(* This function Block interfaces with a NO turbo valve*)
(* Mainly used in the FEE HXR GATT*)
FUNCTION F_TurboExtILK_NO_1 : BOOL
VAR_INPUT
    Turbo		:	ST_PTM;
    BackingGauge:	ST_VG;
    InletGauge	:	ST_VG;
    VentValve	:	ST_VCC_NO; //NO type turbo valve
    ScrollPump	:	ST_RoughPump;
END_VAR

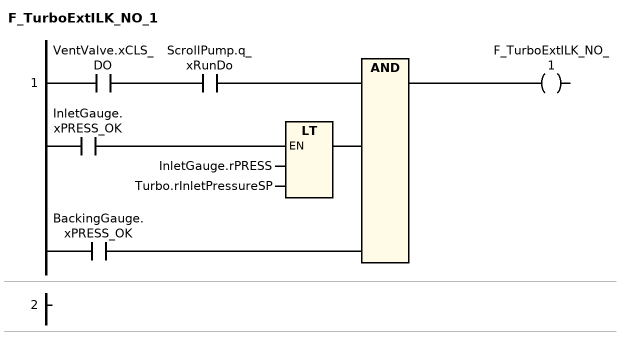
// NETWORK 1
F_TurboExtILK_NO_1 := (VentValve.xCLS_DO AND ScrollPump.q_xRunDo) AND (InletGauge.xPRESS_OK AND InletGauge.rPRESS < Turbo.rInletPressureSP) AND BackingGauge.xPRESS_OK;

// NETWORK 2

END_FUNCTION

(* stored: Version 1.1.0.1
   POU F_TurboExtILK_NO_1: Id {a8dfe7f9-5324-46a7-9f13-de5ec630395c}, SpecialFunc None *)
